FUNCTION_BLOCK speedToRawInt (* Converte a velocidade (%) em valor bruto UINT16 para registrador Modbus *)
  (* Standard: 61499-2 *)
  (* Version 1.0, 10/5/2026, Hidryco, Hidryco, Velocidade em INT para os sopradores Sulzer *)
  PACKAGE SE.Nereda;
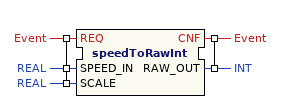
  EVENT_INPUT
    REQ WITH SPEED_IN, SCALE;
  END_EVENT
  EVENT_OUTPUT
    CNF WITH RAW_OUT;
  END_EVENT
  VAR_INPUT
    SPEED_IN : REAL; (* Velocidade em % *)
    SCALE : REAL; (* Fator: valor bruto = % x SCALE *)
  END_VAR
  VAR_OUTPUT
    RAW_OUT : INT; (* Valor bruto (padrao de bits UINT16) *)
  END_VAR
  VAR
    v : REAL;
  END_VAR
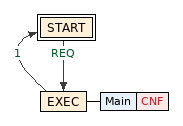
  EC_STATES
    START; (* Initial State *)
    EXEC : Main -> CNF;
  END_STATES
  EC_TRANSITIONS
    START TO EXEC := REQ;
    EXEC TO START := 1;
  END_TRANSITIONS
  ALGORITHM Main IN ST:
(* Referencia de velocidade para registrador de 16 bits (UINT16) do equipamento.
   SPEED_IN em % -> RAW_OUT = SPEED_IN * SCALE, limitado a 0..65535 e entregue como INT
   com o mesmo padrao de bits (valores acima de 32767 viram negativos no INT). *)
v := SPEED_IN * SCALE;
IF v < 0.0 THEN
    v := 0.0;
END_IF;
IF v > 65535.0 THEN
    v := 65535.0;
END_IF;
IF v > 32767.0 THEN
    RAW_OUT := REAL_TO_INT(v - 65536.0);
ELSE
    RAW_OUT := REAL_TO_INT(v);
END_IF;
  END_ALGORITHM
END_FUNCTION_BLOCK
